// TIA Portal V20 export
TYPE "sAxis"
   STRUCT
      I_SS { S7_SetPoint := 'True'} : "sAxis_SS";
      I_CMD { S7_SetPoint := 'True'} : "sAxis_CMD";
      I_Para { S7_SetPoint := 'True'} : "sAxis_Para";
      O_Status { S7_SetPoint := 'True'} : "sAxis_Status";
      I_InLock { S7_SetPoint := 'True'} : "sAxis_InLock";
      I_HMI { S7_SetPoint := 'True'} : "sAxis_HMI";
   END_STRUCT;
END_TYPE
